FUNCTION_BLOCK FINAL GetJsonString IMPLEMENTS Callback
VAR_INPUT
	jsonDomParser: REFERENCE TO FB_JsonDomParser;
	bufferReference: REFERENCE TO STRING(255);
	memberReference: REFERENCE TO SJsonValue;
END_VAR


(* This is method get's exectued by the framework when the callback is triggered.
 It returns a step number which might be used together with Await to jump to a certain chain step
 after the callback code has been executed.*)
METHOD execute : UDINT
bufferReference := jsonDomParser.GetString(memberReference);
END_METHOD

END_FUNCTION_BLOCK

(* stored: Version 1.1.0.1, ProductVersion 3.1.4024.12
   POU GetJsonString: Id {4ec942fc-6682-4887-acc1-e732360b49f2}, SpecialFunc None
   Method execute: Id {3a5a13c9-509b-4412-a403-b76d3ec08e6c} *)
